FUNCTION_BLOCK FB_File
VAR
	fbInfo:			 	FB_FileProperties;
    fbCreateDir:		FB_CreateDir;
	fbOpen:				FB_FileOpen;
	fbRead:				FB_FileRead;
	fbWrite:			FB_FileWrite;
	fbClose:			FB_FileClose;
	fbDelete:			FB_FileDelete;
	pBuffer:			POINTER TO BYTE;
	nBuffer:			UDINT;

END_VAR
VAR_OUTPUT
	bBusy:					BOOL;
	bError:					BOOL;
	nErrId:					UDINT;
END_VAR
VAR CONSTANT
	nMaxFileSize:		UDINT:= 1024 * 1024;
END_VAR

fbInfo();
fbCreateDir();
fbOpen();
fbRead();
fbWrite();
fbClose();
fbDelete();

METHOD PUBLIC M_Append : BOOL
VAR_INPUT
	Text:			STRING(255);
END_VAR
IF fbWrite.bExecute THEN
	IF fbWrite.bError THEN
		nErrId:= fbWrite.nErrId;
		fbWrite.bExecute:= FALSE;
	ELSIF fbWrite.bBusy THEN
		;
	ELSE
		M_Append:= TRUE;
		fbWrite.bExecute:= FALSE;
	END_IF
ELSE
	fbWrite.bExecute:= TRUE;
	fbWrite.pWriteBuff:= ADR(Text);
	fbWrite.cbWriteLen:= INT_TO_UDINT(Len(Text));
END_IF
END_METHOD

METHOD PUBLIC M_Close : BOOL
VAR_INPUT
END_VAR
IF fbClose.bExecute THEN
	IF fbClose.hFile = 0 THEN
		fbClose.bExecute:= FALSE;
		M_Close:= TRUE;
	ELSIF fbClose.bError THEN
		fbClose.bExecute:= FALSE;
		nErrId:= fbClose.nErrId;
	ELSIF fbClose.bBusy THEN
		;
	ELSE
		nErrId:= 0;	
		fbRead.hFile:= 0;
		fbWrite.hFile:= 0;
		fbClose.hFile:= 0;
		fbClose.bExecute:= FALSE;
		M_Close:= TRUE;
	END_IF
ELSE
	fbClose.bExecute:= TRUE;
END_IF
END_METHOD

METHOD PUBLIC M_Create : BOOL
VAR_INPUT
	sPathName:		STRING(255);
END_VAR
VAR
	nTemp: INT;
END_VAR
VAR_INST
	nPosition: INT;
END_VAR
nTemp := FIND(RIGHT(sPathName, LEN(sPathName) - nPosition), '\');
if nTemp <> 0 then
	IF fbCreateDir.bExecute THEN
		IF NOT fbCreateDir.bBusy THEN
			nPosition := nPosition + nTemp;
			fbCreateDir.bExecute:= FALSE;
		END_IF
	ELSE
		fbCreateDir.bExecute:= TRUE;
		fbCreateDir.ePath:= PATH_GENERIC;
		fbCreateDir.sPathName:= Left(sPathName, nPosition + nTemp);
	END_IF
ELSE
	M_Create:= TRUE;
END_IF
END_METHOD

METHOD PUBLIC M_Delete : BOOL
VAR_INPUT
	PathName:		STRING(255);
END_VAR
fbDelete();
IF fbDelete.bExecute THEN
	IF fbDelete.bError THEN
		fbDelete.bExecute:= FALSE;
		M_Delete:= TRUE;
	ELSIF fbDelete.bBusy THEN
		;
	ELSE
		fbDelete.bExecute:= FALSE;
		M_Delete:= TRUE;
	END_IF
ELSE
	fbDelete.bExecute:= TRUE;
	fbDelete.sPathName:= PathName;
	fbDelete.ePath:= E_OpenPath.PATH_GENERIC;
END_IF
END_METHOD

METHOD PUBLIC M_Open : BOOL
VAR_INPUT
	sPathName:		STRING(255);
END_VAR
IF fbOpen.bExecute THEN
	IF fbOpen.bError THEN
		nErrId:= fbOpen.nErrId;
		fbOpen.bExecute:= FALSE;
	ELSIF fbOpen.bBusy THEN
		;
	ELSE
		fbRead.hFile:= fbOpen.hFile;
		fbWrite.hFile:= fbOpen.hFile;
		fbClose.hFile:= fbOpen.hFile;
		fbOpen.bExecute:= FALSE;
		M_Open:= TRUE;
	END_IF	
ELSE
	fbOpen.bExecute:= TRUE;
	fbOpen.sPathName:= sPathName;
	fbOpen.nMode:= (FOPEN_MODEAPPEND OR FOPEN_MODEPLUS OR FOPEN_MODETEXT);
END_IF
END_METHOD

METHOD PUBLIC M_Read : BOOL
VAR_INPUT
	Value:		ANY;
END_VAR
IF fbRead.bExecute THEN
	IF fbRead.bError THEN
		nErrId:= fbRead.nErrId;
		fbRead.bExecute:= FALSE;
	ELSIF fbRead.bBusy THEN
		;
	ELSE
		fbRead.bExecute:= FALSE;
		M_Read:= TRUE;
	END_IF
ELSE
	fbRead.bExecute:= TRUE;
	fbRead.pReadBuff:= pBuffer;
	fbRead.cbReadLen:= nBuffer;
END_IF
END_METHOD

METHOD PUBLIC M_Write : BOOL
VAR_INPUT
	Value:		ANY;
END_VAR
IF fbWrite.bExecute THEN
	IF fbWrite.bError THEN
		nErrId:= fbWrite.nErrId;
		fbWrite.bExecute:= FALSE;
	ELSIF fbWrite.bBusy THEN
		M_Write:= FALSE;
	ELSE
		M_Write:= TRUE;
		fbWrite.bExecute:= FALSE;
	END_IF
ELSE
	fbWrite.bExecute:= TRUE;
	fbRead.pReadBuff:= pBuffer;
	fbRead.cbReadLen:= nBuffer;
END_IF
END_METHOD

END_FUNCTION_BLOCK

(* stored: Version 1.1.0.1
   POU FB_File: Id {54789f62-498b-04f5-3258-42d49534c4a8}, SpecialFunc None
   Method M_Append: Id {1e5af4d0-f329-067d-0bf2-a3973278c0e5}
   Method M_Close: Id {c0789999-930f-042f-18a5-7eb9b96ad755}
   Method M_Create: Id {26efe1d9-595f-0507-2f2f-b4311f718a87}
   Method M_Delete: Id {35d3c0a5-5d24-0db0-05ee-ad42476ea1e5}
   Method M_Open: Id {a8dc81cc-e694-069e-3edb-de6efac1c222}
   Method M_Read: Id {b2e3afdd-1ca1-0d8e-0510-561806c5e056}
   Method M_Write: Id {190fc925-5e69-0b04-04d9-e18614960a32} *)
